INTERFACE ITcoInputDialogFormat

METHOD WithCaption : ITcoInputDialogAnswer
VAR_INPUT
	inCaption : STRING(255);
END_VAR
END_METHOD

METHOD WithImage : ITcoInputDialogAnswer
VAR_INPUT
	inSource : STRING(255);
	inHeight:REAL;
	inWidth:REAL;
END_VAR
END_METHOD

METHOD WithOk : ITcoInputDialogAnswer
VAR_INPUT
END_VAR
END_METHOD

METHOD WithText : ITcoInputDialogAnswer
VAR_INPUT
	inText : STRING(500);
END_VAR
END_METHOD

METHOD WithType : ITcoInputDialogAnswer
VAR_INPUT
	inDialogType : eDialogType;
END_VAR
END_METHOD

METHOD WithYesNo : ITcoInputDialogAnswer
VAR_INPUT
END_VAR
END_METHOD

END_INTERFACE

(* stored: Version 1.1.0.1
   Itf ITcoInputDialogFormat: Id {c5014424-cc29-0e94-1ae6-48b2ac5e9c60}
   Folder Format: Id {34a7c889-714e-0692-32bd-bf4c1ca2eb66}
   Method WithCaption: Id {961cabec-24cf-0fab-2de9-62679dbe5fc5}
   Method WithImage: Id {8fb3da7e-3533-07f9-176e-b2332f5b4ef0}
   Method WithOk: Id {824d6293-b681-07ef-12ab-fb70dd1fa942}
   Method WithText: Id {ffb35f07-c7b9-09a0-160b-7d0019f9f510}
   Method WithType: Id {827d4a98-c60c-0a51-23de-e68a8a9043a0}
   Method WithYesNo: Id {f40f9819-83ad-0754-0917-c963310bb450} *)
